(* IEC 61131-3 sources: POMIRTS_lab3/AS/Library_2/ArUnitText, 3 files *)

(* ---- ArUnitText.typ ---- *)
TYPE
    ARUnitTextTypeEnum :
	(
		arUNITTEXT_SYMBOL		:= 0,
		arUNITTEXT_NAME			:= 1,
		arUNITTEXT_DESCRIPTION	:= 2
	);

	ArUnitTextAsyncInternalType : STRUCT
        FBStateCtx		: ArFBStateInternalType;
		AsyFuMaCtx		: ArFBAsyFuMaInternalType;
	END_STRUCT;

	ArUnitTextGetSymbolInternalType : STRUCT
	    Done					: BOOL;
		Active					: BOOL;
		Busy					: BOOL;
		Error					: BOOL;
		StatusID				: DINT;
		UnitID					: DINT;						(*UnitID of Unit*)
		Namespace				: UDINT;					(*Pointer to String with Namespace of Unit*)
		TextType				: ARUnitTextTypeEnum;		(*Type of Text (Symbol, Name, ...)*)
		ResultText				: UDINT;					(*Pointer to String with resulting Unit Symbol*)
		ResultSize				: UDINT;					(*Max Length of SymbolString*)
		UseBRText				: BOOL;						(*Use text from B&R as default*)
		LanguageCode			: STRING[18];				(*LanguageCode*)
		TextSize				: UDINT;					(*Length of text in result-buffer*)
		ExecuteOld				: BOOL;
	END_STRUCT;

	ArUnitTextCCToUIDInternalType : STRUCT
		Done					: BOOL;
		Active					: BOOL;
		Busy					: BOOL;
		Error					: BOOL;
		ErrorID					: DINT;
		CommonCode				: STRING[3];	(*CommonCode*)
		UnitID					: DINT;
		ExecuteOld				: BOOL;
	END_STRUCT;

END_TYPE

(* ---- ArUnitText.fun ---- *)
{REDUND_CONTEXT} {REDUND_UNREPLICABLE} FUNCTION_BLOCK ArUnitTextGetText		(*Get text of units.*)
	VAR_INPUT
		Execute				: BOOL;						(*Start execution.*)
		UnitID				: DINT;						(*Identifier of unit.*)
		Namespace			: UDINT;					(*Pointer to a string with the namespace of the unit, 0 for default namespace.*)
		TextType			: ARUnitTextTypeEnum;		(*Type of text (Symbol, Name, ...).*)
		ResultText			: UDINT;					(*Pointer to the buffer to which the resulting text is copied.*)
		ResultSize			: UDINT;					(*Maximal length of resulting text.*)
		UseBRText			: BOOL;						(*Use unit text from B+R namespace as default.*)
		LanguageCode		: STRING[18];				(*Language code (eg. en, de).*)
	END_VAR
	VAR_OUTPUT
		Done				: BOOL; 					(*Execution done.*)
		Busy				: BOOL; 					(*Execution running.*)
		Error				: BOOL; 					(*Execution failed.*)
		StatusID			: DINT;						(*Execution error: see help.*)
		TextSize			: UDINT;					(*Length of text copied into result buffer.*)
	END_VAR
	VAR
        Internal			: ArUnitTextAsyncInternalType;		(*Internal variable.*)
	END_VAR
END_FUNCTION_BLOCK

{REDUND_CONTEXT} {REDUND_UNREPLICABLE} FUNCTION_BLOCK ArUnitTextCommonCodeToUnitID		(*Converts the common code of an unit to its identifier.*)
	VAR_INPUT
		Execute			: BOOL;				(*Start execution.*)
		CommonCode		: STRING[3];		(*Common code.*)
	END_VAR
	VAR_OUTPUT
		Done					: BOOL;		(*Execution done.*)
		Busy					: BOOL;     (*Execution running.*)
		Error					: BOOL;     (*Execution failed.*)
		StatusID		 		: DINT;	    (*Execution error: see help.*)
		UnitID					: DINT;     (*Unit identifier.*)
	END_VAR
	VAR
        Internal				: ArUnitTextAsyncInternalType;		(*Internal variable.*)
	END_VAR
END_FUNCTION_BLOCK

(* ---- ArUnitText.var ---- *)
VAR CONSTANT
	arUNITTEXT_ERR_NO_TEXT_FOUND		: DINT := -1070585646;			(*Text not found.*)
	arUNITTEXT_ERR_INVALID_CC			: DINT := -1070585645;          (*Invalid common code.*)
	arUNITTEXT_ERR_INVALID_PARAM		: DINT := -1070585644;          (*Invalid parameter.*)
	arUNITTEXT_ERR_INTERNAL				: DINT := -1070585643;          (*An internal error has occurred. Please contact B+R support.*)
	arUNITTEXT_OK_USER_TEXT				: DINT := 3156178;              (*Resulting text is from user namespace.*)
	arUNITTEXT_OK_BR_TEXT				: DINT := 3156179;              (*Resulting text is from B+R default namespace.*)
END_VAR
